// TIA Portal V18 export
TYPE "ModeOutStruct"
// stored: IsFailsafeCompliant false
   STRUCT
      Estop : Bool;   // 急停
      Reset : Bool;   // 复位
      Manual : Bool;   // 手动
      Auto : Bool;   // 自动
      Home : Bool;   // 回原位
      Running : Bool;   // 运行中
      Change : Bool;   // 模式变化
   END_STRUCT;
END_TYPE
